Staubli VAL3: Alter.pgx

program Alter()
begin
  wait(bAlterRun == true and isSettled() == false)
  nAlterBegin=alterBegin(world,mAlterspeed)

  while nAlterBegin>=0 and bAlterRun==true
    if bAlterRun==true
      trOffset.x = 0
      trOffset.y = 0
      trOffset.z = nDeltZ
      trOffset.rx = 0
      trOffset.ry = 0
      trOffset.rz = 0
    elseIf bAlterRun==false
      trOffset.z = 0
    endIf
    nAlter = alter(trOffset)
      delay(0.004)
  endWhile
end
